// TIA Portal V17 export
// export: Created 2025-03-10T13:11:58.9053587Z, ExportSetting WithDefaults, DisplayName Totally Integrated Automation Portal, DisplayVersion V17 Update 8, DisplayName TIA Portal Openness, DisplayVersion V17 Update 8, DisplayName TIA Portal Version Control Interface, DisplayVersion V17, DisplayName SINAMICS Startdrive Advanced, DisplayVersion V17 SP2, DisplayName SINAMICS Startdrive G110M, G120, G120C, G120D, G120P, G115D, DisplayVersion V17 SP2, DisplayName SINAMICS Startdrive G130, G150, S120, S150, SINAMICS MV, S210, DisplayVersion V17 SP2, DisplayName STEP 7 Professional, DisplayVersion V17 Update 8, DisplayName SINUMERIK ONE STEP 7 Toolbox, DisplayVersion V17 Update 12, DisplayName SINUMERIK 840D sl STEP 7 Toolbox, DisplayVersion V17 Update 12, DisplayName STEP 7 Safety, DisplayVersion V17 Update 6, DisplayName WinCC Advanced, DisplayVersion V17 Update 8
TYPE "LBP_typeMcp483StandardInput"
TITLE = MCP 483 image / Imagen de MCP 483 / MCP 483 Abbild
// Input image of MCP 483 / Imagen de entrada de MCP 483 / Eingangsabbild von MCP 483
// stored: IsFailsafeCompliant false
   STRUCT
      auto : Bool;
      mda : Bool;
      teachIn : Bool;
      jog : Bool;
      spindleOvrA : Bool;
      spindleOvrB : Bool;
      spindleOvrC : Bool;
      spindleOvrD : Bool;
      inc1 : Bool;
      inc10 : Bool;
      inc100 : Bool;
      inc1000 : Bool;
      inc10000 : Bool;
      incVar : Bool;
      refPoint : Bool;
      repos : Bool;
      cycleStop : Bool;
      cycleStart : Bool;
      feedrateStop : Bool;
      feedrateStart : Bool;
      spindleStop : Bool;
      spindleStart : Bool;
      keySwitch2 : Bool;
      keySwitch0 : Bool;
      feedrateOvrA : Bool;
      feedrateOvrB : Bool;
      feedrateOvrC : Bool;
      feedrateOvrD : Bool;
      feedrateOvrE : Bool;
      singleBlock : Bool;
      keySwitch1 : Bool;
      reset : Bool;
      axis10 : Bool;   // R10
      axis7 : Bool;   // R7
      axis4 : Bool;   // R4
      axisX : Bool;   // R1
      keySwitch3 : Bool;
      rapidTraverse : Bool;   // R14
      minus : Bool;   // R13
      plus : Bool;   // R15
      axis6 : Bool;   // R6
      axis8 : Bool;   // R8
      axis9 : Bool;   // R9
      axis11 : Bool;   // R11
      mcsWcs : Bool;   // R12
      axis5 : Bool;   // R5
      axisZ : Bool;   // R3
      axisY : Bool;   // R2
      reserved60 : Bool;
      customerKey15 : Bool;   // T15
      customerKey14 : Bool;   // T14
      customerKey13 : Bool;   // T13
      customerKey12 : Bool;   // T12
      customerKey11 : Bool;   // T11
      customerKey10 : Bool;   // T10
      customerKey9 : Bool;   // T9
      customerKey8 : Bool;   // T8
      customerKey7 : Bool;   // T7
      customerKey6 : Bool;   // T6
      customerKey5 : Bool;   // T5
      customerKey4 : Bool;   // T4
      customerKey3 : Bool;   // T3
      customerKey2 : Bool;   // T2
      customerKey1 : Bool;   // T1
   END_STRUCT;
END_TYPE
